// TwinCAT 3 PLC project getData
// ProgramVersion: 3.1.4020.4
// libraries:
//   Tc2_Standard, * (Beckhoff Automation GmbH)
//   Tc2_System, * (Beckhoff Automation GmbH)
//   Tc3_Module, * (Beckhoff Automation GmbH)
// project tree:
//   / PlcTask.TcTTO
//   POUs/ MAIN.TcPOU
// real-time tasks:
//   TASK PlcTask: cycle T#10ms, priority 20, ADS port 350
// motion (NC):
//   TASK NC-Task 1 SAF: cycle T#2ms, priority 4, ADS port 501
//   TASK NC-Task 1 SVB: cycle T#10ms, priority 8, ADS port 511
//   AXIS Axis 1 (id 1)
//     Dynamic: AccelerationMaximum=450000, DecelerationMaximum=450000, Acceleration=5566, Deceleration=5566, Jerk=5566
//     Velo: SlowManual=50000, FastManual=100000, Maximum=150000
//     PositionAreaControl: Enable=false, RefSearch=false
//     TargetPosControl: Enable=false
//     OtherSettings: AllowMotionCmdToSlave=true
//     encoder EncType=19
//       EncPara: ScaleFactorNumerator=1, MaxCount=#xffffffff
//     drive DrvType=16
//       DrvPara: MaxCount=#xffffffff
//         Analog: VeloReferenz=150000
//         TimeComp: TaskDelayCycles=1
//     controller CtrType=1
//       CtrPara: PriorControlFactor=1
//         PosDiffControl: Enable=false
//         Observer: BandWidth=20
// I/O:
//   DEVICE Device 3 (EtherCAT), AmsNetId 172.18.138.230.4.1
//     Drive 1 (ZeroErr Driver) [ZeroErr Driver]
// variable links:
//   NC-Task 1 SAF/Axes/Axis 1 <-> Device 3 (EtherCAT)/Drive 1 (ZeroErr Driver)
//     Drive/Inputs/In/nDcOutputTime <-> InfoData/DcOutputShift
//     Drive/Inputs/In/nState1 <-> Transmit PDO mapping 0/Status word
//     Drive/Inputs/In/nState2 <-> Transmit PDO mapping 0/Status word @bit 8
//     Drive/Inputs/In/nState4 @bit 1 <-> WcState/InputToggle
//     Drive/Inputs/In/nState4 <-> WcState/WcState
//     Drive/Outputs/Out/nCtrl1 <-> Receive PDO mapping 0/Control word
//     Drive/Outputs/Out/nCtrl2 <-> Receive PDO mapping 0/Control word @bit 8
//     Drive/Outputs/Out/nDataOut1 <-> Receive PDO mapping 0/Target Position
//     Enc/Inputs/In/nDataIn1 <-> Transmit PDO mapping 0/Position actual value
//     Enc/Inputs/In/nDcInputTime <-> InfoData/DcInputShift
//     Enc/Inputs/In/nState4 @bit 1 <-> WcState/InputToggle
//     Enc/Inputs/In/nState4 <-> WcState/WcState
//   getData/getData Instance <-> Device 3 (EtherCAT)/Drive 1 (ZeroErr Driver)
//     PlcTask Inputs/MAIN.DualPosDiff <-> Transmit PDO mapping 0/Dual encoder difference value
//     PlcTask Inputs/MAIN.actPosition <-> Transmit PDO mapping 0/Position actual value_1
//     PlcTask Inputs/MAIN.actVelo <-> Transmit PDO mapping 0/Actual velocity
//     PlcTask Outputs/MAIN.siOperationMode <-> Receive PDO mapping 0/Modes of operation
//     PlcTask Outputs/MAIN.targetVelo <-> Receive PDO mapping 0/Target Velocity
//     PlcTask Outputs/MAIN.udiProAcc <-> Receive PDO mapping 0/Profile acceleration
//     PlcTask Outputs/MAIN.udiProDec <-> Receive PDO mapping 0/Profile deceleration

CONFIGURATION getData
    RESOURCE PLC ON TwinCAT3
        TASK PlcTask(INTERVAL := T#10ms, PRIORITY := 20);
        PROGRAM MAIN WITH PlcTask : MAIN;
    END_RESOURCE
END_CONFIGURATION

// ---- POUs/MAIN.TcPOU
PROGRAM MAIN
VAR
	(*--- Triansmit PDO ---*)
	DualPosDiff       AT%I*   :DINT;//双编码器差值
	actVelo           AT%I*   :DINT;//实际速度
	actPosition       AT%I*   :DINT;//实际位置
	(*--- Receive PDO ---*)
	targetVelo        AT%Q*   :DINT;//目标速度
	siOperationMode   AT%Q*   :SINT;//运动模式
	udiProAcc         AT%Q*   :UDINT;//目标加速度
	udiProDec         AT%Q*   :UDINT;//目标减速度
	(*--- User ---*)
	modAngle:     DINT;//角度取余
	actAngle:     LREAL;//实际角度
	rotation        :BOOL;//旋转方向
	rotationSingle  :INT;//旋转标志位
	sampleVelo:   DINT;
END_VAR

siOperationMode := 3;
udiProAcc:=50000;
udiProDec:=50000;
//计算当前角度
modAngle:= ABS(actPosition MOD 524288);//角度取余
actAngle:= (DINT_TO_LREAL(modAngle)/524288)*360;//实际角度
IF rotation = FALSE THEN
	IF actAngle < 180 THEN
		IF rotationSingle = 2 THEN//切换模式
			rotation := TRUE;
			rotationSingle := 3;
			targetVelo:=0;
		ELSE
			IF actAngle <= 5 THEN
				rotationSingle := 1;
			END_IF
			targetVelo:=(ABS(LREAL_TO_DINT(actAngle*1.5)))+30;
		END_IF	
	ELSIF actAngle >= 180 THEN
		IF actAngle >= 355 AND rotationSingle = 1 THEN
			rotationSingle := 2;
		END_IF
		targetVelo:=(ABS(LREAL_TO_DINT((360-actAngle)*1.5)))+30;
	END_IF
ELSE 
	IF actAngle < 180 THEN
		IF actAngle <= 5 AND rotationSingle = 4 THEN
			rotationSingle := 5;
		END_IF
		targetVelo:=-(ABS(LREAL_TO_DINT(actAngle*1.5)))-30;
	ELSIF actAngle >= 180 THEN
		IF rotationSingle = 5 THEN//切换模式
			rotation := 0;
			rotationSingle := 0;
			targetVelo:=0;
		ELSE
			IF actAngle >= 355 THEN
				rotationSingle := 4;
			END_IF
			targetVelo:=-(ABS(LREAL_TO_DINT((360-actAngle)*1.5)))-30;
		END_IF	
	END_IF
END_IF
sampleVelo := targetVelo * 257;

END_PROGRAM
